// TIA Portal V17 export
// export: Created 2022-07-16T16:56:22.8916576Z, ExportSetting WithDefaults, DisplayName Totally Integrated Automation Portal, DisplayVersion V17, DisplayName TIA Portal Openness, DisplayVersion V17, DisplayName TIA Portal Version Control Interface, DisplayVersion V17, DisplayName TIA Portal Test Suite Advanced, DisplayVersion V17, DisplayName STEP 7 Professional, DisplayVersion V17, DisplayName STEP 7 Safety, DisplayVersion V17, DisplayName WinCC Professional, DisplayVersion V17
TYPE "udtOtherPressure"
// stored: IsFailsafeCompliant false
   STRUCT
      avaragePressure : Int;
      tripleValidationActive : Int;
      dualValidationActive : Int;
      pressure1failed : Bool;
      pressure2failed : Bool;
      pressure3failed : Bool;
      moreThen1pressureFailed : Bool;
   END_STRUCT;
END_TYPE
